FUNCTION_BLOCK FB_FifoIndexer
VAR_INPUT
    MaxSize : UDINT;  // Set once, e.g., in init
	EnableWrapAround : BOOL := FALSE;	// Enable wrap-around when buffer is full
END_VAR
VAR_OUTPUT
END_VAR
VAR
    _readIndex : UDINT := 0;
    _writeIndex : UDINT := 0;
    _count : UDINT := 0;
END_VAR

PROPERTY Count : UDINT
GET
Count := _count;
END_GET
END_PROPERTY

METHOD Dequeue : BOOL;
VAR_INPUT
END_VAR
IF IsEmpty THEN 
	Dequeue := FALSE; // Empty
	RETURN;
END_IF

Dequeue := TRUE;
_readIndex := (_readIndex + 1) MOD MaxSize;
_count := _count - 1;
END_METHOD

METHOD Enqueue : BOOL;
VAR_INPUT
END_VAR
IF IsFull AND NOT EnableWrapAround THEN
	Enqueue := FALSE; // Full
	RETURN;
END_IF

Enqueue := TRUE;
_writeIndex := (_writeIndex + 1) MOD MaxSize;
_count := _count + 1;
END_METHOD

PROPERTY IsEmpty : BOOL
GET
IsEmpty := (_readIndex = _writeIndex) AND (_count = 0);
END_GET
END_PROPERTY

PROPERTY IsFull : BOOL
GET
IsFull := _writeIndex = _readIndex AND _count = MaxSize;
END_GET
END_PROPERTY

PROPERTY ReadIndex : UDINT
GET
ReadIndex := _readIndex;
END_GET
END_PROPERTY

PROPERTY WriteIndex : UDINT
GET
WriteIndex := _writeIndex;
END_GET
END_PROPERTY

END_FUNCTION_BLOCK

(* stored: Version 1.1.0.1
   POU FB_FifoIndexer: Id {d166dc60-92bf-4432-a19b-528d3364e3d7}, SpecialFunc None
   Property Count: Id {e7524c59-89f9-43b3-bdac-091ca75407f8}
   Get Get: Id {7175b43f-9c26-4fb2-8eda-caa1c8958d9e}
   Method Dequeue: Id {1304ba0c-e2f2-44e9-9436-d63b0b9ec44c}
   Method Enqueue: Id {536852e1-aa18-4cf3-bfee-13736057a888}
   Property IsEmpty: Id {262bf447-955a-4423-adae-e1817d4940e8}
   Get Get: Id {6f4a96bf-173f-435e-8cb4-0017ef5c0d5d}
   Property IsFull: Id {d562d59b-ee88-46ca-b8bb-26d311f7f704}
   Get Get: Id {34e06915-e3a4-4ce6-8fe7-b0f1d8ce0412}
   Property ReadIndex: Id {2a58dc7d-a5ba-4338-afbe-8a860dc76c71}
   Get Get: Id {b6b0c5a0-0039-407a-95dd-39d25078bafb}
   Property WriteIndex: Id {ee8c5686-5e93-4042-a1e6-eaaeec5dee9c}
   Get Get: Id {d1f17506-a9dc-4142-b1a2-07fd4646582b} *)
